FUNCTION BisscEvaluator : ST_BeamDemand
VAR_INPUT
	encoder : ST_BisscEncoder;
END_VAR
VAR	
	readLoc: ULINT;
	newDemand : ST_BeamDemand;
END_VAR

readLoc := Encoder.encLoc;
IF readLoc <= Encoder.ncULimit THEN
	newDemand.demand := TRUE;
ELSE
	newDemand.demand := FALSE;
END_IF

IF readLoc <= Encoder.ncULimit THEN 
	newDemand.beamRate := 0;
ELSE
	newDemand.beamRate := 50;
END_IF

BisscEvaluator := newDemand;

END_FUNCTION

(* stored: Version 1.1.0.1, ProductVersion 3.1.4020.12
   POU BisscEvaluator: Id {0cb3e4b3-8172-46ac-8d55-9c1f5efc80d4}, SpecialFunc None *)
